gfCNCPoint1[29987] = {X 202.4356, Y 18.3712, Z -2.1667, A 0.000, B 0.000, C 0.000 }
gfCNCPoint1[29988] = {X 202.7123, Y 20.0435, Z -2.1667, A 0.000, B 0.000, C 0.000 }
gfCNCPoint1[29989] = {X 202.7957, Y 21.7363, Z -2.1667, A 0.000, B 0.000, C 0.000 }
gfCNCPoint1[29990] = {X 202.6848, Y 23.4277, Z -2.1667, A 0.000, B 0.000, C 0.000 }
gfCNCPoint1[29991] = {X 202.3810, Y 25.0952, Z -2.1667, A 0.000, B 0.000, C 0.000 }
gfCNCPoint1[29992] = {X 201.9139, Y 26.6019, Z -2.1667, A 0.000, B 0.000, C 0.000 }
gfCNCPoint1[29993] = {X 201.2442, Y 28.0301, Z -2.1667, A 0.000, B 0.000, C 0.000 }
gfCNCPoint1[29994] = {X 200.3845, Y 29.3527, Z -2.1667, A 0.000, B 0.000, C 0.000 }
gfCNCPoint1[29995] = {X 199.3512, Y 30.5446, Z -2.1667, A 0.000, B 0.000, C 0.000 }
gfCNCPoint1[29996] = {X 198.1639, Y 31.5832, Z -2.1667, A 0.000, B 0.000, C 0.000 }
gfCNCPoint1[29997] = {X 199.0622, Y 31.8618, Z -2.1667, A 0.000, B 0.000, C 0.000 }
gfCNCPoint1[29998] = {X 199.8728, Y 32.3386, Z -2.1667, A 0.000, B 0.000, C 0.000 }
gfCNCPoint1[29999] = {X 200.5527, Y 32.9884, Z -2.1667, A 0.000, B 0.000, C 0.000 }
gfCNCPoint1[30000] = {X 201.0657, Y 33.7766, Z -2.1667, A 0.000, B 0.000, C 0.000 }

ENDDAT
